(* Logix 5000 project; controller Prueba2 vendor 1 type 14 code 156 rev 30.11; software revision 30.00 *)

TASK MainTask (continuous, watchdog 500 ms) : MainProgram

MODULES
   Local : vendor 1 type 14 code 156 (Compact 0, rev 30.11)
      DI_4 : 1769-IQ16 (Compact 4, rev 1.1, Input RPI 20 ms)
      DO_5 : vendor 1 type 7 code 86 (Compact 5, rev 2.1, Output RPI 20 ms)
END_MODULES

ADD_ON_INSTRUCTION ACT_DE   (* revision 1.0 *)
VAR_INPUT
   PRENDER_DE : BOOL; {required}
   CIERRE_DE : BOOL; {access None, required}
END_VAR
VAR_OUTPUT
   APERTURA_DE : BOOL; {access None, required}
END_VAR
VAR
   TON_APERTURA_DE : TIMER := (PRE := 1000); {access None}
   E_PRENDER : BOOL;
END_VAR

ROUTINE Logic   (* ladder *)
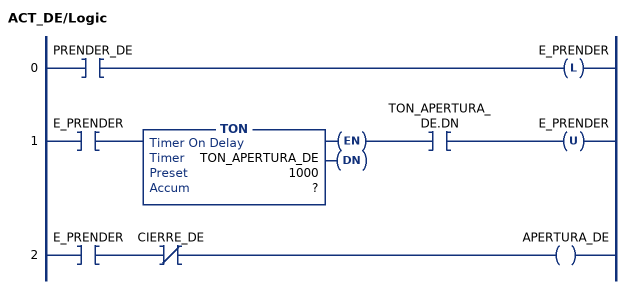
   0: XIC(PRENDER_DE)OTL(E_PRENDER);
   1: XIC(E_PRENDER)TON(TON_APERTURA_DE,?,?)XIC(TON_APERTURA_DE.DN)OTU(E_PRENDER);
   2: XIC(E_PRENDER)XIO(CIERRE_DE)OTE(APERTURA_DE);
END_ROUTINE
END_ADD_ON_INSTRUCTION

ADD_ON_INSTRUCTION CIE_DE   (* revision 1.0 *)
VAR_INPUT
   APAGAR_DE : BOOL; {required}
   APERTURA_DE : BOOL; {required}
END_VAR
VAR_OUTPUT
   CIERRE_DE : BOOL; {access Read Only, required}
END_VAR
VAR
   E_APAGAR : BOOL; {access None}
   TON_CIERRE_dE : TIMER := (PRE := 300); {access None}
END_VAR

ROUTINE Logic   (* ladder *)
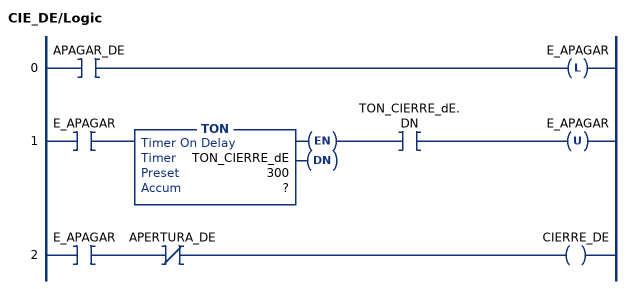
   0: XIC(APAGAR_DE)OTL(E_APAGAR);
   1: XIC(E_APAGAR)TON(TON_CIERRE_dE,?,?)XIC(TON_CIERRE_dE.DN)OTU(E_APAGAR);
   2: XIC(E_APAGAR)XIO(APERTURA_DE)OTE(CIERRE_DE);
END_ROUTINE
END_ADD_ON_INSTRUCTION

VAR_GLOBAL   (* controller tags *)
   ACT_SE : ACT_DE;
   APAGAR_DE : BOOL;
   APERTURA_DE : ALIAS FOR Local:5:O.Data.4;
   APERTURA_SE : ALIAS FOR Local:5:O.Data.6;
   CIERRE_DE : ALIAS FOR Local:5:O.Data.5;
   Count_S1 : COUNTER := (PRE := 3);
   E_APAGAR : BOOL;
   E_PRENDER : BOOL;
   GD_IN_0 : BOOL;
   GD_IN_1 : BOOL;
   GD_IN_2 : BOOL;   // GD sensor 1
   GD_IN_3 : BOOL := 1;
   GD_IN_4 : BOOL;
   GD_IN_5 : BOOL;   // GD RESET
   GD_OUT_0 : BOOL;
   GD_OUT_1 : BOOL;
   PRENDER_DE : BOOL;
   PRENDER_SE : BOOL;
   Prueba_1 : ACT_DE;
   PRUEBA_2 : CIE_DE;
   SENSOR : BOOL;
   TagA : BOOL;
   TB1 : BOOL;
   TB2 : BOOL;
   TIMER1 : TIMER := (PRE := 5000);
   TON_APERTURA_DE : TIMER := (PRE := 300);
   TON_CIERRE_dE : TIMER := (PRE := 300);
END_VAR

PROGRAM MainProgram   (* main routine MainRoutine *)
VAR
   PS_BANDA1 : ALIAS FOR Local:5:O.Data.0;
   PS_START : ALIAS FOR Local:4:I.Data.1;
   PS_STOP : ALIAS FOR Local:4:I.Data.0;
END_VAR

ROUTINE MainRoutine   (* ladder *)
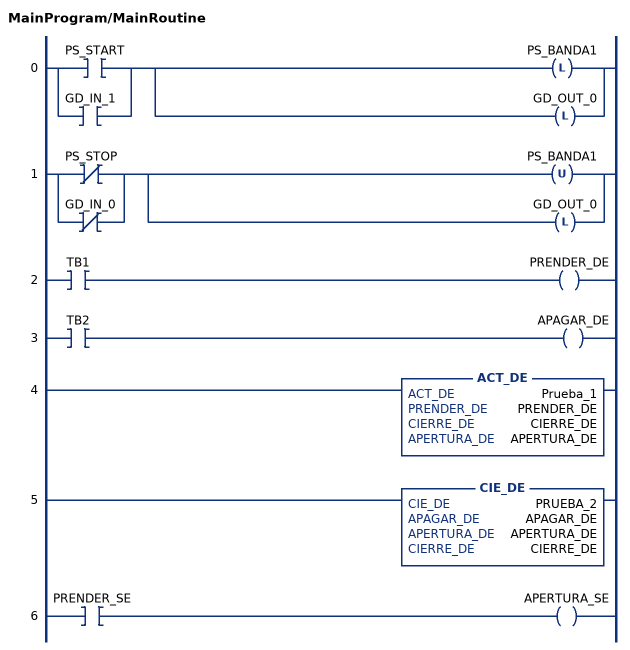
   0: [XIC(PS_START) ,XIC(GD_IN_1) ][OTL(PS_BANDA1) ,OTL(GD_OUT_0) ];
   1: [XIO(PS_STOP) ,XIO(GD_IN_0) ][OTU(PS_BANDA1) ,OTL(GD_OUT_0) ];
   2: XIC(TB1)OTE(PRENDER_DE);
   3: XIC(TB2)OTE(APAGAR_DE);
   4: ACT_DE(Prueba_1,PRENDER_DE,CIERRE_DE,APERTURA_DE);
   5: CIE_DE(PRUEBA_2,APAGAR_DE,APERTURA_DE,CIERRE_DE);
   6: XIC(PRENDER_SE)OTE(APERTURA_SE);
END_ROUTINE
END_PROGRAM
